// TwinCAT 3 PLC project Twincat_Utulities
// ProgramVersion: 3.1.4023.0
// libraries:
//   Tc2_Standard, * (Beckhoff Automation GmbH)
//   Tc2_System, * (Beckhoff Automation GmbH)
//   Tc2_Utilities, * (Beckhoff Automation GmbH)
//   Tc3_Module, * (Beckhoff Automation GmbH)
// project tree:
//   DUTs/ E_EventType.TcDUT (not stored), ST_Event.TcDUT (not stored)
//   / PlcTask.TcTTO
//   POUs/ EventBuffer.TcPOU, MAIN.TcPOU, TestFuntionBlock.TcPOU
// real-time tasks:
//   TASK PlcTask: cycle T#10ms, priority 20, ADS port 350

CONFIGURATION Twincat_Utulities
    RESOURCE PLC ON TwinCAT3
        TASK PlcTask(INTERVAL := T#10ms, PRIORITY := 20);
        PROGRAM MAIN WITH PlcTask : MAIN;
    END_RESOURCE
END_CONFIGURATION

// ---- POUs/MAIN.TcPOU
PROGRAM MAIN
VAR
	Event_Buffer : EventBuffer;
	
	addEvent : BOOL;
	addEvent2 :BOOL;
	stEventToAdd :ST_Event;
	bEventToAddError : BOOL;
	
	
	ReadAndRemoved_Event : BOOL;
    ReadAndRemoved_Event2 : BOOL;
	stLastReadEvent: ST_Event;
	stLastReadEvent2: ST_Event;
	bReadAndRemoveEventError : BOOL;
END_VAR


IF AddEvent THEN 
	Event_Buffer.AddEvent(st_Event:= stEventToAdd, bError =>	bEventToAddError );
	addEvent := FALSE;
END_IF

IF ReadAndRemoved_Event THEN 
	
	Event_Buffer.ReadAndRemoveEvent(stEvent => stLastReadEvent, bError =>	bReadAndRemoveEventError );
	ReadAndRemoved_Event := FALSE;
END_IF

END_PROGRAM

// ---- POUs/EventBuffer.TcPOU
FUNCTION_BLOCK EventBuffer
VAR
	MemRingBuffer : FB_MemRingBuffer ;
	BufferArray  : ARRAY[0..MAX_BUFFER_SIZE] OF BYTE; (* Buffer memory used by FB_MemRingBuffer function block *)
END_VAR

VAR CONSTANT 
	 MAX_BUFFER_SIZE : UDINT := 1000;
	 SIZE_OF_ST_EVENT : UDINT := SIZEOF(ST_Event);
	 MAX_NUMBER_OF_ST_EVENT : UDINT := 5;
	 NUMBER_OF_BYTES_FOR_ALL_ST_EVENT: UDINT := SIZE_OF_ST_EVENT *  MAX_NUMBER_OF_ST_EVENT;
	 	
END_VAR

METHOD PUBLIC AddEvent
VAR_INPUT
	st_Event : REFERENCE TO  ST_Event ;
	
END_VAR

VAR_OUTPUT
	bError : BOOL;
END_VAR
MemRingBuffer.A_AddTail(pWrite := ADR(st_Event),
	                    cbWrite := SIZEOF(st_Event),
						pBuffer := ADR(BufferArray),
						cbBuffer := SIZEOF(BufferArray));

						
bError := NOT MemRingBuffer.bOk;
END_METHOD

METHOD PUBLIC ReadAndRemoveEvent
VAR_OUTPUT
	stEvent	: ST_Event;
	bError : BOOL;
END_VAR
MemRingBuffer.A_RemoveHead(pRead := ADR(stEvent),
	                       cbRead := SIZEOF(stEvent),
						   pBuffer := ADR(BufferArray),
						   cbBuffer := SIZEOF(BufferArray));

						
bError := NOT MemRingBuffer.bOk;
END_METHOD

END_FUNCTION_BLOCK

// ---- POUs/TestFuntionBlock.TcPOU
FUNCTION_BLOCK TestFuntionBlock
VAR
	nCounter : LINT;
	
END_VAR

nCounter := nCounter +1;

END_FUNCTION_BLOCK
